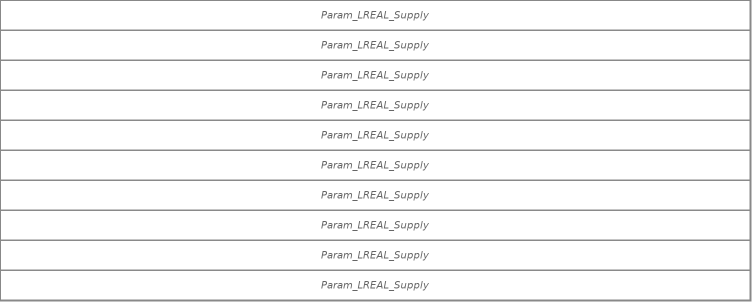
VISUALIZATION Visu_Supply_Params  // 752x302
    Frame (0,0 750x30)
        shows Param_LREAL_Supply(nIdx := GlobalOne)
    Frame (0,30 750x30)
        shows Param_LREAL_Supply(nIdx := 2)
    Frame (0,60 750x30)
        shows Param_LREAL_Supply(nIdx := 3)
    Frame (0,120 750x30)
        shows Param_LREAL_Supply(nIdx := 5)
    Frame (0,90 750x30)
        shows Param_LREAL_Supply(nIdx := 4)
    Frame (0,270 750x30)
        shows Param_LREAL_Supply(nIdx := 10)
    Frame (0,240 750x30)
        shows Param_LREAL_Supply(nIdx := 9)
    Frame (0,210 750x30)
        shows Param_LREAL_Supply(nIdx := 8)
    Frame (0,180 750x30)
        shows Param_LREAL_Supply(nIdx := 7)
    Frame (0,150 750x30)
        shows Param_LREAL_Supply(nIdx := 6)
END_VISUALIZATION

(* stored: Version 1.1.0.1, ProductVersion 3.1.4024.12
   Visu Visu_Supply_Params: Id {e7bedc7a-015c-4a2e-a2b7-b3635c7b51d3} *)
